SUBAPPLICATION mapping_Buttons (* Subapplication Type *)
  (* Standard: 61499-2 *)
  (* Version 1.0, 2023-01-29, Franz *)
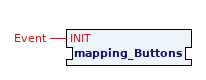
  EVENT_INPUT
    INIT;
  END_EVENT
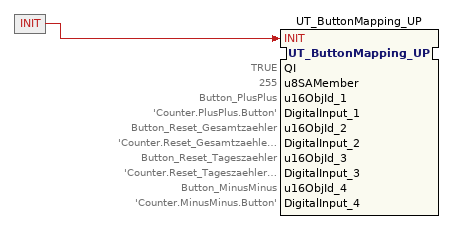
  FBS
    UT_ButtonMapping_UP : UT_ButtonMapping_UP(QI := TRUE, u8SAMember := 255, u16ObjId_1 := Button_PlusPlus, DigitalInput_1 := 'Counter.PlusPlus.Button', u16ObjId_2 := Button_Reset_Gesamtzaehler, DigitalInput_2 := 'Counter.Reset_Gesamtzaehler.Button', u16ObjId_3 := Button_Reset_Tageszaehler, DigitalInput_3 := 'Counter.Reset_Tageszaehler.Button', u16ObjId_4 := Button_MinusMinus, DigitalInput_4 := 'Counter.MinusMinus.Button');
  END_FBS
  EVENT_CONNECTIONS
    INIT TO UT_ButtonMapping_UP.INIT;
  END_CONNECTIONS
END_SUBAPPLICATION
